// TIA Portal V16 export
// export: Created 2022-07-21T09:35:17.3514937Z, ExportSetting WithDefaults, DisplayName Totally Integrated Automation Portal, DisplayVersion V16 Update 4, DisplayName TIA Portal Version Control Interface, DisplayVersion V16 Update 2, DisplayName TIA Portal Openness, DisplayVersion V16 Update 4, DisplayName SINAMICS Startdrive Advanced, DisplayVersion V16 Update 5, DisplayName SINAMICS Startdrive G130, G150, S120, S150, SINAMICS MV, S210, DisplayVersion V16 Update 5, DisplayName SINAMICS Startdrive G110M, G120, G120C, G120D, G120P, G115D, DisplayVersion V16 Update 5, DisplayName STEP 7 Professional, DisplayVersion V16 Update 4, DisplayName STEP 7 Safety, DisplayVersion V16, DisplayName WinCC Advanced, DisplayVersion V16 Update 4
DATA_BLOCK "dbLotCode"   // DB1
{ S7_Optimized_Access := 'TRUE' }
VERSION : 0.1
// stored: AutoNumber true, DBAccessibleFromOPCUA true, IsOnlyStoredInLoadMemory false, IsRetainMemResEnabled false, IsWriteProtectedInAS false, MemoryReserve 100
   VAR
      Product_TR300 : Array[1..10] of Struct
         SKU : String;
         Code : String;
      END_STRUCT;
      Product_ADFLO : Array[1..10] of Struct
         SKU : String;
         Code : String;
      END_STRUCT;
   END_VAR
BEGIN
   Product_TR300[1].SKU := 'SKU: 7100018971';
   Product_TR300[2].SKU := 'SKU: 7100019023';
   Product_TR300[3].SKU := 'SKU: 7100018972';
   Product_TR300[4].SKU := 'SKU: 7100018965';
   Product_TR300[1..3].Code := '3712U';
   Product_TR300[4].Code := '3712E';
   Product_ADFLO[1].SKU := 'SKU: 7000118083';
   Product_ADFLO[2].SKU := 'SKU: 7100116817';
   Product_ADFLO[3].SKU := 'SKU: 7100057907';
   Product_ADFLO[4].SKU := 'SKU: 7100057889';
   Product_ADFLO[1].Code := 'ADU';
   Product_ADFLO[2..4].Code := 'ADE';
END_DATA_BLOCK
